% RSLogix 500 project P4_ABIOLA_A_V11_BAK100.RSS, saved by version 8.30.00.16 %
PROJECT "UNTITLED"    % processor: Bul.1763 MicroLogix 1100 Series B %

PROGRAM FILES
  LAD 2   4 rungs
  LAD 3 "INPUTS"  6 rungs  % This contains all input instructions used.   %
  LAD 4 "OUTPUTS"  2 rungs  % This contains all output instructions %
  LAD 5 "PRO LOGIC"  14 rungs  % This contains all the logic instructions used  %

DATA FILES
  O0 OUTPUT  4 elements
  I1 INPUT  6 elements
  S2 STATUS  66 elements
  B3 BINARY  1 elements
  T4 TIMER  4 elements
  C5 COUNTER  2 elements
  R6 CONTROL  1 elements
  N7 INTEGER  2 elements
  F8 FLOAT  1 elements

LADDER 2
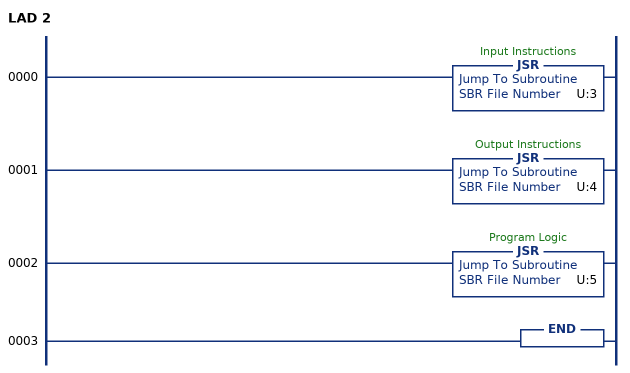
% Rung: 0 %
SOR JSR U:3 EOR
%   U:3  "Input Instructions" %
% Rung: 1 %
SOR JSR U:4 EOR
%   U:4  "Output Instructions" %
% Rung: 2 %
SOR JSR U:5 EOR
%   U:5  "Program Logic" %
% Rung: 3 %
SOR END EOR

LADDER 3 "INPUTS"    % This contains all input instructions used.   %
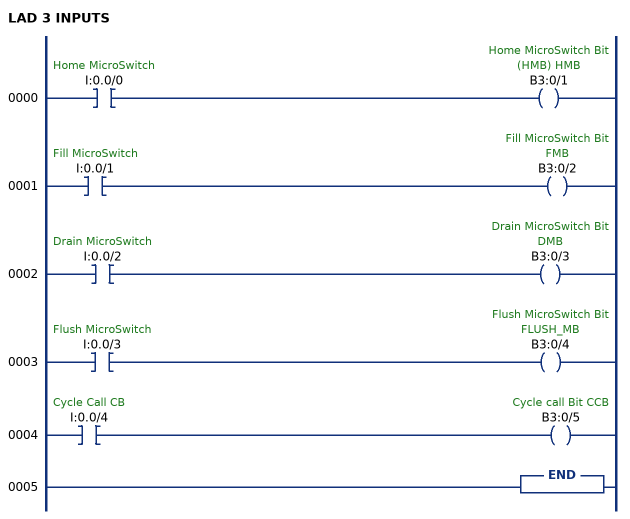
% Rung: 0 %
SOR XIC I:0.0/0 OTE B3:0/1 EOR
%   I:0.0/0  "Home MicroSwitch" %
%   B3:0/1  HMB  "Home MicroSwitch Bit (HMB)" %
% Rung: 1 %
SOR XIC I:0.0/1 OTE B3:0/2 EOR
%   I:0.0/1  "Fill MicroSwitch" %
%   B3:0/2  FMB  "Fill MicroSwitch Bit" %
% Rung: 2 %
SOR XIC I:0.0/2 OTE B3:0/3 EOR
%   I:0.0/2  "Drain MicroSwitch" %
%   B3:0/3  DMB  "Drain MicroSwitch Bit" %
% Rung: 3 %
SOR XIC I:0.0/3 OTE B3:0/4 EOR
%   I:0.0/3  "Flush MicroSwitch" %
%   B3:0/4  FLUSH_MB  "Flush MicroSwitch Bit" %
% Rung: 4 %
SOR XIC I:0.0/4 OTE B3:0/5 EOR
%   I:0.0/4  CB  "Cycle Call" %
%   B3:0/5  CCB  "Cycle call Bit" %
% Rung: 5 %
SOR END EOR

LADDER 4 "OUTPUTS"    % This contains all output instructions %
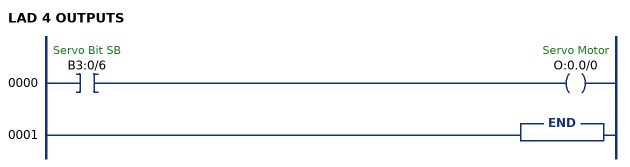
% Rung: 0 %
SOR XIC B3:0/6 OTE O:0.0/0 EOR
%   B3:0/6  SB  "Servo Bit" %
%   O:0.0/0  "Servo Motor" %
% Rung: 1 %
SOR END EOR

LADDER 5 "PRO LOGIC"    % This contains all the logic instructions used  %
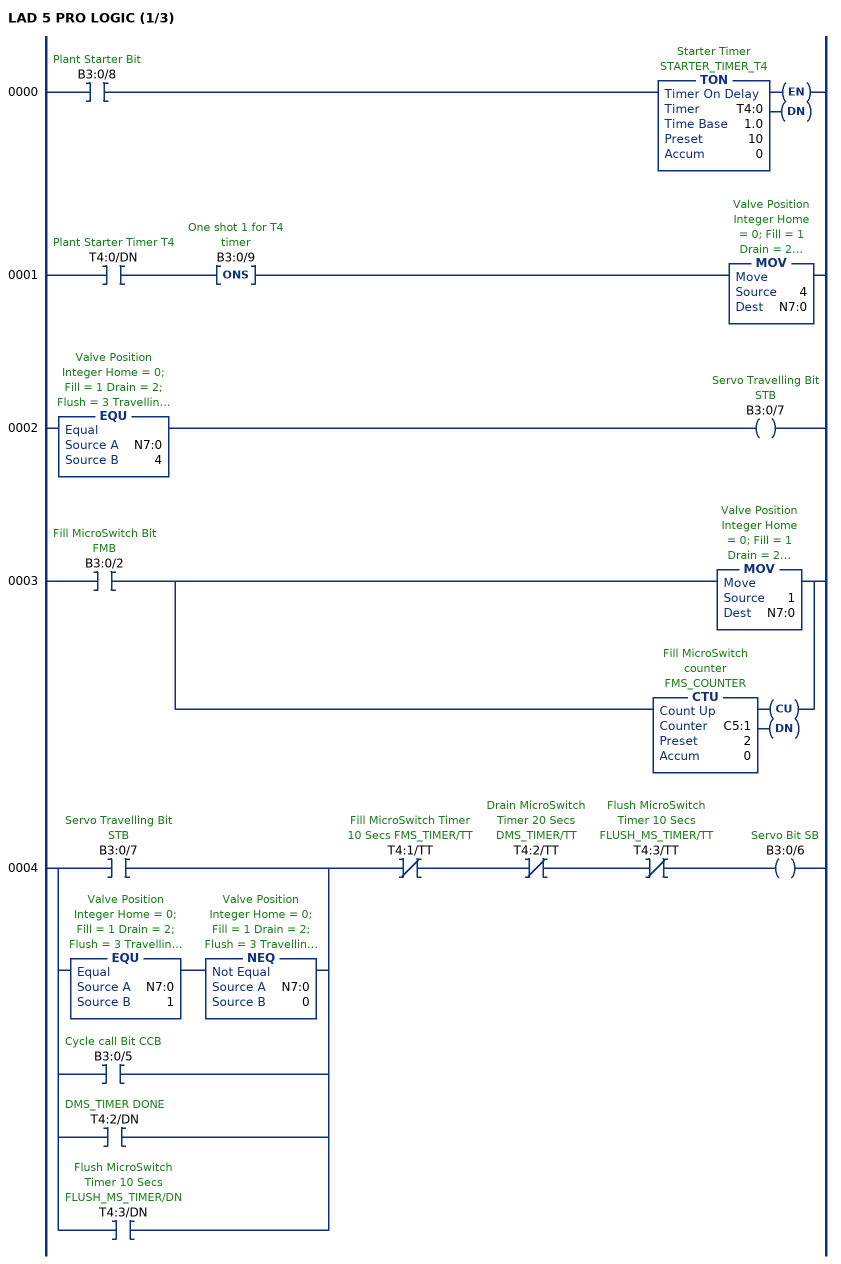
% Rung: 0 %
SOR XIC B3:0/8 TON T4:0 1.0 10 0 EOR
%   B3:0/8  "Plant Starter Bit" %
%   T4:0  STARTER_TIMER_T4  "Starter Timer" %
% Rung: 1 %
SOR XIC T4:0/DN ONS B3:0/9 MOV 4 N7:0 EOR
%   T4:0/DN  T4  "Plant Starter Timer" %
%   B3:0/9  "One shot 1 for T4 timer" %
%   N7:0  VALVE_PI  "Valve Position Integer Home = 0; Fill = 1 Drain = 2; Flush = 3 Travelling = 4" %
% Rung: 2 %
SOR EQU N7:0 4 OTE B3:0/7 EOR
%   N7:0  VALVE_PI  "Valve Position Integer Home = 0; Fill = 1 Drain = 2; Flush = 3 Travelling = 4" %
%   B3:0/7  STB  "Servo Travelling Bit" %
% Rung: 3 %
SOR XIC B3:0/2 BST MOV 1 N7:0 NXB CTU C5:1 2 0 BND EOR
%   B3:0/2  FMB  "Fill MicroSwitch Bit" %
%   N7:0  VALVE_PI  "Valve Position Integer Home = 0; Fill = 1 Drain = 2; Flush = 3 Travelling = 4" %
%   C5:1  FMS_COUNTER  "Fill MicroSwitch counter" %
% Rung: 4 %
SOR BST XIC B3:0/7 NXB BST EQU N7:0 1 NEQ N7:0 0 NXB BST XIC B3:0/5 NXB BST XIC T4:2/DN NXB XIC T4:3/DN BND BND BND BND XIO T4:1/TT XIO T4:2/TT XIO T4:3/TT OTE B3:0/6 EOR
%   B3:0/7  STB  "Servo Travelling Bit" %
%   N7:0  VALVE_PI  "Valve Position Integer Home = 0; Fill = 1 Drain = 2; Flush = 3 Travelling = 4" %
%   B3:0/5  CCB  "Cycle call Bit" %
%   T4:2/DN  "DMS_TIMER DONE" %
%   T4:3  FLUSH_MS_TIMER  "Flush MicroSwitch Timer 10 Secs" %
%   T4:1  FMS_TIMER  "Fill MicroSwitch Timer 10 Secs" %
%   T4:2  DMS_TIMER  "Drain MicroSwitch Timer 20 Secs" %
%   B3:0/6  SB  "Servo Bit" %

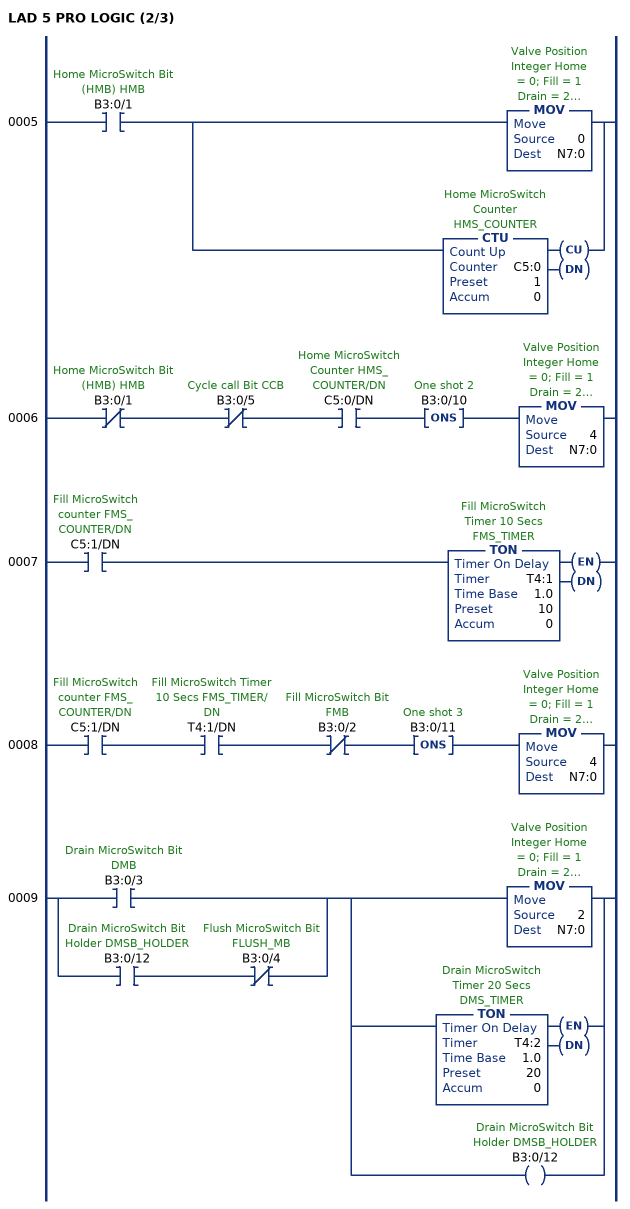
% Rung: 5 %
SOR XIC B3:0/1 BST MOV 0 N7:0 NXB CTU C5:0 1 0 BND EOR
%   B3:0/1  HMB  "Home MicroSwitch Bit (HMB)" %
%   N7:0  VALVE_PI  "Valve Position Integer Home = 0; Fill = 1 Drain = 2; Flush = 3 Travelling = 4" %
%   C5:0  HMS_COUNTER  "Home MicroSwitch Counter" %
% Rung: 6 %
SOR XIO B3:0/1 XIO B3:0/5 XIC C5:0/DN ONS B3:0/10 MOV 4 N7:0 EOR
%   B3:0/1  HMB  "Home MicroSwitch Bit (HMB)" %
%   B3:0/5  CCB  "Cycle call Bit" %
%   C5:0  HMS_COUNTER  "Home MicroSwitch Counter" %
%   B3:0/10  "One shot 2" %
%   N7:0  VALVE_PI  "Valve Position Integer Home = 0; Fill = 1 Drain = 2; Flush = 3 Travelling = 4" %
% Rung: 7 %
SOR XIC C5:1/DN TON T4:1 1.0 10 0 EOR
%   C5:1  FMS_COUNTER  "Fill MicroSwitch counter" %
%   T4:1  FMS_TIMER  "Fill MicroSwitch Timer 10 Secs" %
% Rung: 8 %
SOR XIC C5:1/DN XIC T4:1/DN XIO B3:0/2 ONS B3:0/11 MOV 4 N7:0 EOR
%   C5:1  FMS_COUNTER  "Fill MicroSwitch counter" %
%   T4:1  FMS_TIMER  "Fill MicroSwitch Timer 10 Secs" %
%   B3:0/2  FMB  "Fill MicroSwitch Bit" %
%   B3:0/11  "One shot 3" %
%   N7:0  VALVE_PI  "Valve Position Integer Home = 0; Fill = 1 Drain = 2; Flush = 3 Travelling = 4" %
% Rung: 9 %
SOR BST XIC B3:0/3 NXB XIC B3:0/12 XIO B3:0/4 BND BST MOV 2 N7:0 NXB BST TON T4:2 1.0 20 0 NXB OTE B3:0/12 BND BND EOR
%   B3:0/3  DMB  "Drain MicroSwitch Bit" %
%   B3:0/12  DMSB_HOLDER  "Drain MicroSwitch Bit Holder" %
%   B3:0/4  FLUSH_MB  "Flush MicroSwitch Bit" %
%   N7:0  VALVE_PI  "Valve Position Integer Home = 0; Fill = 1 Drain = 2; Flush = 3 Travelling = 4" %
%   T4:2  DMS_TIMER  "Drain MicroSwitch Timer 20 Secs" %

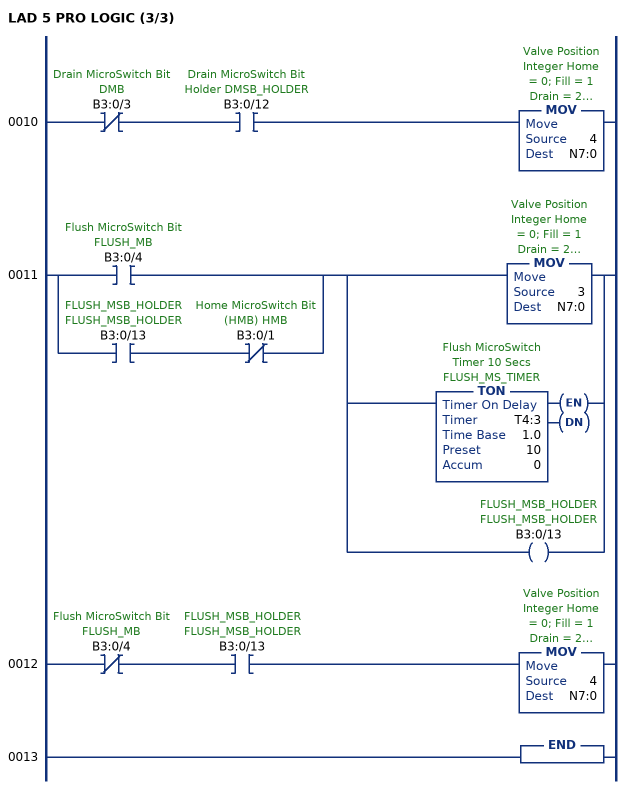
% Rung: 10 %
SOR XIO B3:0/3 XIC B3:0/12 MOV 4 N7:0 EOR
%   B3:0/3  DMB  "Drain MicroSwitch Bit" %
%   B3:0/12  DMSB_HOLDER  "Drain MicroSwitch Bit Holder" %
%   N7:0  VALVE_PI  "Valve Position Integer Home = 0; Fill = 1 Drain = 2; Flush = 3 Travelling = 4" %
% Rung: 11 %
SOR BST XIC B3:0/4 NXB XIC B3:0/13 XIO B3:0/1 BND BST MOV 3 N7:0 NXB BST TON T4:3 1.0 10 0 NXB OTE B3:0/13 BND BND EOR
%   B3:0/4  FLUSH_MB  "Flush MicroSwitch Bit" %
%   B3:0/13  FLUSH_MSB_HOLDER  "FLUSH_MSB_HOLDER" %
%   B3:0/1  HMB  "Home MicroSwitch Bit (HMB)" %
%   N7:0  VALVE_PI  "Valve Position Integer Home = 0; Fill = 1 Drain = 2; Flush = 3 Travelling = 4" %
%   T4:3  FLUSH_MS_TIMER  "Flush MicroSwitch Timer 10 Secs" %
% Rung: 12 %
SOR XIO B3:0/4 XIC B3:0/13 MOV 4 N7:0 EOR
%   B3:0/4  FLUSH_MB  "Flush MicroSwitch Bit" %
%   B3:0/13  FLUSH_MSB_HOLDER  "FLUSH_MSB_HOLDER" %
%   N7:0  VALVE_PI  "Valve Position Integer Home = 0; Fill = 1 Drain = 2; Flush = 3 Travelling = 4" %
% Rung: 13 %
SOR END EOR

OTHER DOCUMENTED ADDRESSES
  N7:1  AC_CYCLE_BIT  "Active state on Cycle bit"

DATA TABLE (non-zero values as saved)
DATA T4
% .PRE .ACC %
% T4:0 % 10 0
% T4:1 % 10 0
% T4:2 % 20 0
% T4:3 % 10 0
DATA C5
% .PRE .ACC %
% C5:0 % 1 0
% C5:1 % 2 0
